{attribute 'GeneratedUsingTerminal: AX8108-0100-0101-0101'}
{attribute addProperty BoxType "AX8108-0100-0101-0101"}
{attribute addProperty Id "FSOEAT %I*FSOE_31BB7F2A21"}
{attribute addProperty CRC "856307172"}
{attribute addProperty Size "21"}
TYPE FSoE_Slave_Connection_1_Slave_Message_330A35E4 :
STRUCT
	{attribute addProperty Name "FSOE"}
	FSOE AT %I* : FSOE_31BB7F2A;
END_STRUCT
END_TYPE

(* stored: Version 1.2.0.0, ProductVersion 3.1.4024.9
   DUT FSoE_Slave_Connection_1_Slave_Message_330A35E4: Id {b227515a-9650-4bd4-a420-054e302ed228} *)
